(* IEC 61131-3 sources: CodesysTest/export/Function Blocks/IO/FB_PhysicalDigitalInput.pou/IsOn.prop, 1 file *)

(* ---- Get.pm.st ---- *)
(*#-#-#-#-#-#-#-#-#-#---Declaration---#-#-#-#-#-#-#-#-#-#-#-#-#*)

VAR
END_VAR
(*#-#-#-#-#-#-#-#-#-#---Implementation---#-#-#-#-#-#-#-#-#-#-#-#-#*)

IsOn := Active;
